// TIA Portal V18 export
FUNCTION "potlife&regenaration" : Void   // FC22, LAD
{ S7_Optimized_Access := 'TRUE' }
VERSION : 0.1
// stored: AutoNumber true, IsIECCheckEnabled false, SetENOAutomatically false, UDAEnableTagReadback false
   VAR_TEMP
      temp2 : Bool;
   END_VAR
   VAR_TEMP   // added for the SCL form of the ladder/FBD networks
      _w1 : Bool;
   END_VAR
BEGIN

REGION Network 1: regeneration selection
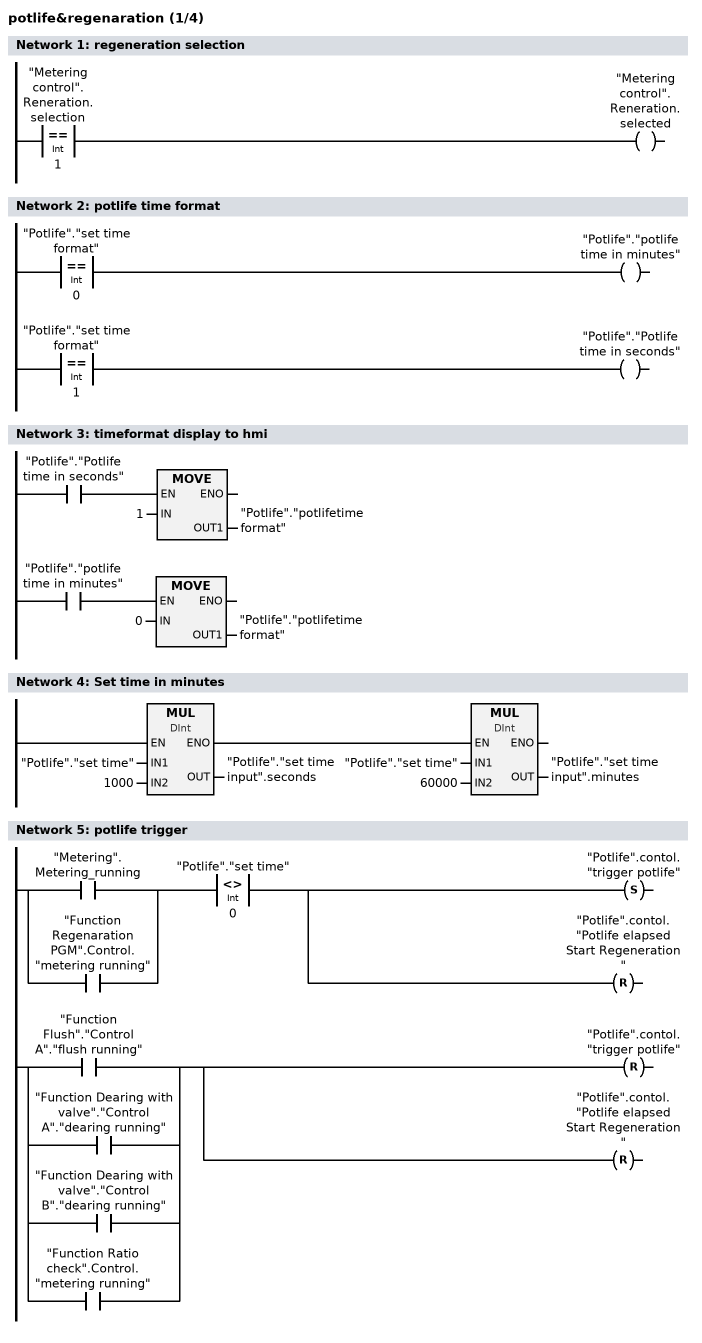
   RUNG wire#powerrail
      { S7_Templates := "SrcType := Int" } EQ_Contact(in1 := "Metering control".Reneration.selection, in2 := 1)
      Coil( "Metering control".Reneration.selected )
   END_RUNG
   // the same network as SCL:
   "Metering control".Reneration.selected := "Metering control".Reneration.selection = 1;
END_REGION

REGION Network 2: potlife time format
   RUNG wire#powerrail
      { S7_Templates := "SrcType := Int" } EQ_Contact(in1 := "Potlife"."set time format", in2 := 0)
      Coil( "Potlife"."potlife time in minutes" )
   END_RUNG
   RUNG wire#powerrail
      { S7_Templates := "SrcType := Int" } EQ_Contact(in1 := "Potlife"."set time format", in2 := 1)
      Coil( "Potlife"."Potlife time in seconds" )
   END_RUNG
   // the same network as SCL:
   "Potlife"."potlife time in minutes" := "Potlife"."set time format" = 0;
   "Potlife"."Potlife time in seconds" := "Potlife"."set time format" = 1;
END_REGION

REGION Network 3: timeformat display to hmi
   RUNG wire#powerrail
      Contact( "Potlife"."Potlife time in seconds" )
      Move(in := 1, out1 => "Potlife"."potlifetime format")
   END_RUNG
   RUNG wire#powerrail
      Contact( "Potlife"."potlife time in minutes" )
      Move(in := 0, out1 => "Potlife"."potlifetime format")
   END_RUNG
   // the same network as SCL:
   IF "Potlife"."Potlife time in seconds" THEN "Potlife"."potlifetime format" := 1; END_IF;
   IF "Potlife"."potlife time in minutes" THEN "Potlife"."potlifetime format" := 0; END_IF;
END_REGION

REGION Network 4: Set time in minutes
   RUNG wire#powerrail
      { S7_Templates := "SrcType := DInt" } Mul(in1 := "Potlife"."set time", in2 := 1000, out => "Potlife"."set time input".seconds)
      { S7_Templates := "SrcType := DInt" } Mul(in1 := "Potlife"."set time", in2 := 60000, out => "Potlife"."set time input".minutes)
   END_RUNG
   // the same network as SCL:
   "Potlife"."set time input".seconds := "Potlife"."set time" * 1000;
   "Potlife"."set time input".minutes := "Potlife"."set time" * 60000;
END_REGION

REGION Network 5: potlife trigger
   RUNG wire#powerrail
      Contact( "Metering".Metering_running )
      wire#w1
      { S7_Templates := "SrcType := Int" } NE_Contact(in1 := "Potlife"."set time", in2 := 0)
      wire#w2
      S_Coil( "Potlife".contol."trigger potlife" )
   END_RUNG
   RUNG wire#powerrail
      Contact( "Function Regenaration PGM".Control."metering running" )
   END_RUNG wire#w1
   RUNG wire#w2
      R_Coil( "Potlife".contol."Potlife elapsed Start Regeneration" )
   END_RUNG
   RUNG wire#powerrail
      Contact( "Function Flush"."Control A"."flush running" )
      wire#w3
      R_Coil( "Potlife".contol."trigger potlife" )
   END_RUNG
   RUNG wire#powerrail
      Contact( "Function Dearing with valve"."Control A"."dearing running" )
   END_RUNG wire#w3
   RUNG wire#powerrail
      Contact( "Function Dearing with valve"."Control B"."dearing running" )
   END_RUNG wire#w3
   RUNG wire#powerrail
      Contact( "Function Ratio check".Control."metering running" )
   END_RUNG wire#w3
   RUNG wire#w3
      R_Coil( "Potlife".contol."Potlife elapsed Start Regeneration" )
   END_RUNG
   // the same network as SCL:
   IF ("Metering".Metering_running OR "Function Regenaration PGM".Control."metering running") AND ("Potlife"."set time" <> 0) THEN
       "Potlife".contol."trigger potlife" := TRUE;
       "Potlife".contol."Potlife elapsed Start Regeneration" := FALSE;
   END_IF;
   IF "Function Flush"."Control A"."flush running" OR "Function Dearing with valve"."Control A"."dearing running" OR "Function Dearing with valve"."Control B"."dearing running" OR "Function Ratio check".Control."metering running" THEN
       "Potlife".contol."trigger potlife" := FALSE;
       "Potlife".contol."Potlife elapsed Start Regeneration" := FALSE;
   END_IF;
END_REGION

REGION Network 6
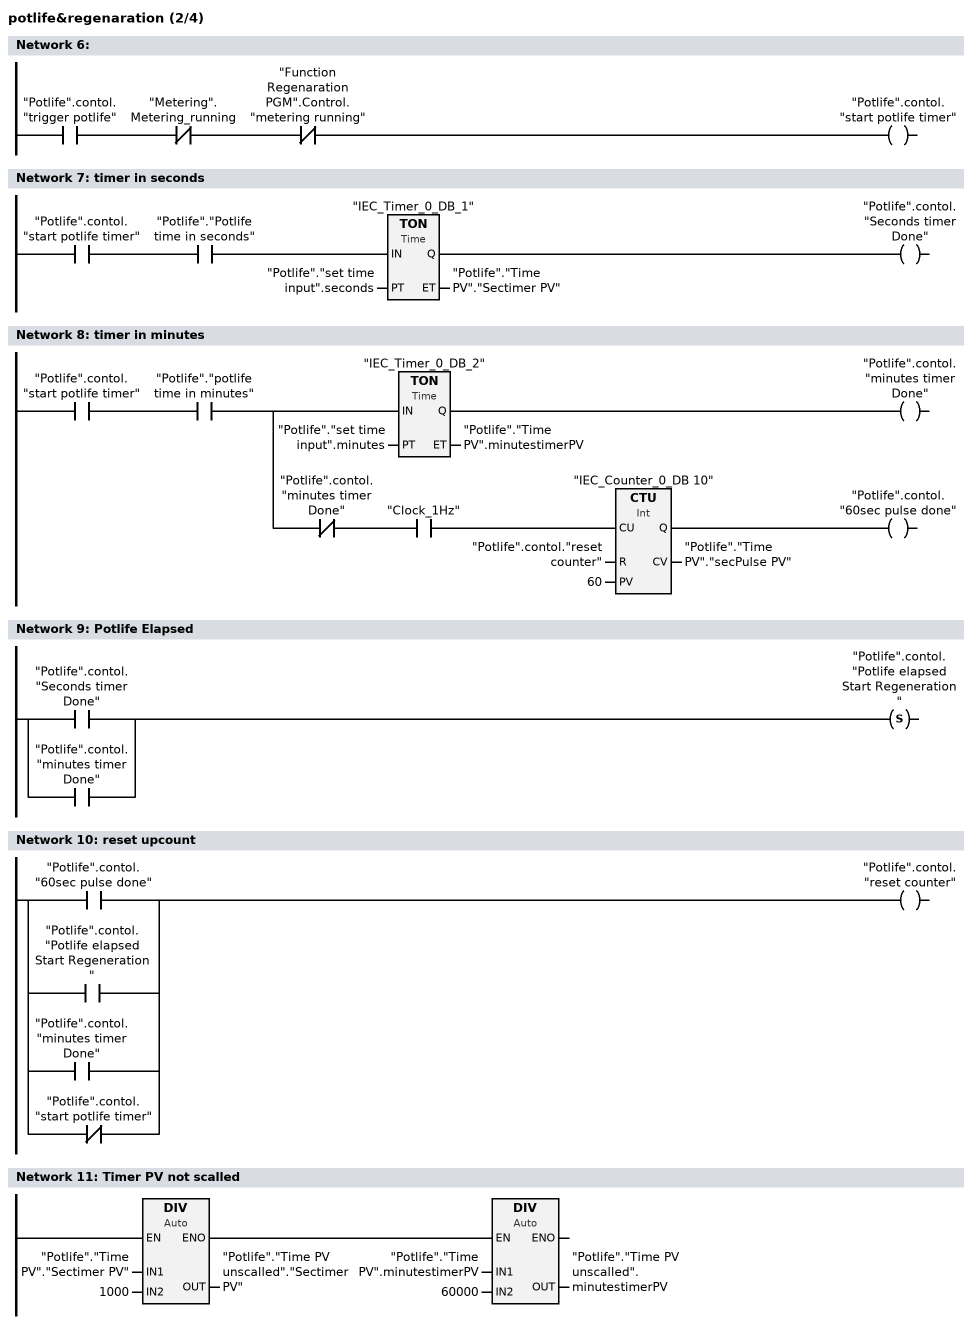
   RUNG wire#powerrail
      Contact( "Potlife".contol."trigger potlife" )
      I_Contact( "Metering".Metering_running )
      I_Contact( "Function Regenaration PGM".Control."metering running" )
      Coil( "Potlife".contol."start potlife timer" )
   END_RUNG
   // the same network as SCL:
   "Potlife".contol."start potlife timer" := "Potlife".contol."trigger potlife" AND NOT "Metering".Metering_running AND NOT "Function Regenaration PGM".Control."metering running";
END_REGION

REGION Network 7: timer in seconds
   RUNG wire#powerrail
      Contact( "Potlife".contol."start potlife timer" )
      Contact( "Potlife"."Potlife time in seconds" )
      { S7_Templates := "time_type := Time" } "IEC_Timer_0_DB_1".TON(pt := "Potlife"."set time input".seconds, et => "Potlife"."Time PV"."Sectimer PV")
      Coil( "Potlife".contol."Seconds timer Done" )
   END_RUNG
   // the same network as SCL:
   "IEC_Timer_0_DB_1".TON(IN := "Potlife".contol."start potlife timer" AND "Potlife"."Potlife time in seconds",
                          PT := "Potlife"."set time input".seconds,
                          ET => "Potlife"."Time PV"."Sectimer PV");
   "Potlife".contol."Seconds timer Done" := "IEC_Timer_0_DB_1".Q;
END_REGION

REGION Network 8: timer in minutes
   RUNG wire#powerrail
      Contact( "Potlife".contol."start potlife timer" )
      Contact( "Potlife"."potlife time in minutes" )
      wire#w1
      { S7_Templates := "time_type := Time" } "IEC_Timer_0_DB_2".TON(pt := "Potlife"."set time input".minutes, et => "Potlife"."Time PV".minutestimerPV)
      Coil( "Potlife".contol."minutes timer Done" )
   END_RUNG
   RUNG wire#w1
      I_Contact( "Potlife".contol."minutes timer Done" )
      Contact( "Clock_1Hz" )
      { S7_Templates := "value_type := Int" } "IEC_Counter_0_DB 10".CTU(r := "Potlife".contol."reset counter", pv := 60, cv => "Potlife"."Time PV"."secPulse PV")
      Coil( "Potlife".contol."60sec pulse done" )
   END_RUNG
   // the same network as SCL:
   #_w1 := "Potlife".contol."start potlife timer" AND "Potlife"."potlife time in minutes";
   "IEC_Timer_0_DB_2".TON(IN := #_w1,
                          PT := "Potlife"."set time input".minutes,
                          ET => "Potlife"."Time PV".minutestimerPV);
   "Potlife".contol."minutes timer Done" := "IEC_Timer_0_DB_2".Q;
   "IEC_Counter_0_DB 10".CTU(CU := #_w1 AND NOT "Potlife".contol."minutes timer Done" AND "Clock_1Hz",
                           R := "Potlife".contol."reset counter",
                           PV := 60,
                           CV => "Potlife"."Time PV"."secPulse PV");
   "Potlife".contol."60sec pulse done" := "IEC_Counter_0_DB 10".Q;
END_REGION

REGION Network 9: Potlife Elapsed
   RUNG wire#powerrail
      Contact( "Potlife".contol."Seconds timer Done" )
      wire#w1
      S_Coil( "Potlife".contol."Potlife elapsed Start Regeneration" )
   END_RUNG
   RUNG wire#powerrail
      Contact( "Potlife".contol."minutes timer Done" )
   END_RUNG wire#w1
   // the same network as SCL:
   IF "Potlife".contol."Seconds timer Done" OR "Potlife".contol."minutes timer Done" THEN
       "Potlife".contol."Potlife elapsed Start Regeneration" := TRUE;
   END_IF;
END_REGION

REGION Network 10: reset upcount
   RUNG wire#powerrail
      Contact( "Potlife".contol."60sec pulse done" )
      wire#w1
      Coil( "Potlife".contol."reset counter" )
   END_RUNG
   RUNG wire#powerrail
      Contact( "Potlife".contol."Potlife elapsed Start Regeneration" )
   END_RUNG wire#w1
   RUNG wire#powerrail
      Contact( "Potlife".contol."minutes timer Done" )
   END_RUNG wire#w1
   RUNG wire#powerrail
      I_Contact( "Potlife".contol."start potlife timer" )
   END_RUNG wire#w1
   // the same network as SCL:
   "Potlife".contol."reset counter" := "Potlife".contol."60sec pulse done" OR "Potlife".contol."Potlife elapsed Start Regeneration" OR "Potlife".contol."minutes timer Done" OR NOT "Potlife".contol."start potlife timer";
END_REGION

REGION Network 11: Timer PV not scalled
   RUNG wire#powerrail
      Div(in1 := "Potlife"."Time PV"."Sectimer PV", in2 := 1000, out => "Potlife"."Time PV unscalled"."Sectimer PV")
      Div(in1 := "Potlife"."Time PV".minutestimerPV, in2 := 60000, out => "Potlife"."Time PV unscalled".minutestimerPV)
   END_RUNG
   // the same network as SCL:
   "Potlife"."Time PV unscalled"."Sectimer PV" := "Potlife"."Time PV"."Sectimer PV" / 1000;
   "Potlife"."Time PV unscalled".minutestimerPV := "Potlife"."Time PV".minutestimerPV / 60000;
END_REGION

REGION Network 12: run time down count
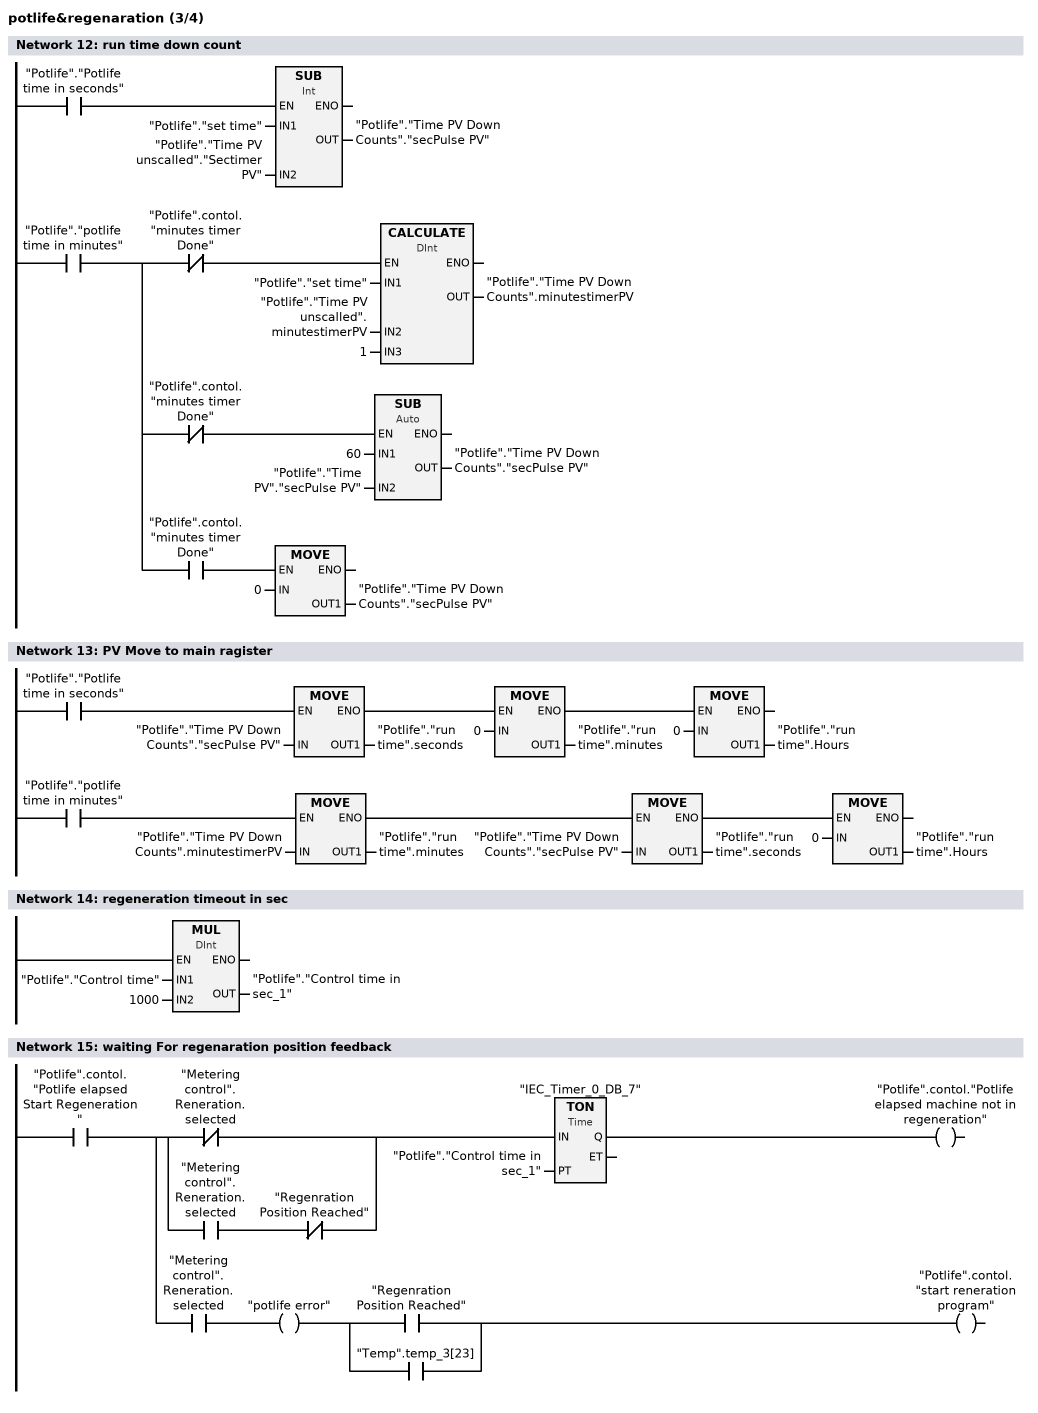
   RUNG wire#powerrail
      Contact( "Potlife"."Potlife time in seconds" )
      { S7_Templates := "SrcType := Int" } Sub(in1 := "Potlife"."set time", in2 := "Potlife"."Time PV unscalled"."Sectimer PV", out => "Potlife"."Time PV Down Counts"."secPulse PV")
   END_RUNG
   RUNG wire#powerrail
      Contact( "Potlife"."potlife time in minutes" )
      wire#w1
      I_Contact( "Potlife".contol."minutes timer Done" )
      { S7_Templates := "SrcType := DInt"; S7_Expression := "IN1-IN2-IN3" } Calculate(in1 := "Potlife"."set time", in2 := "Potlife"."Time PV unscalled".minutestimerPV, in3 := 1, out => "Potlife"."Time PV Down Counts".minutestimerPV)
   END_RUNG
   RUNG wire#w1
      I_Contact( "Potlife".contol."minutes timer Done" )
      Sub(in1 := 60, in2 := "Potlife"."Time PV"."secPulse PV", out => "Potlife"."Time PV Down Counts"."secPulse PV")
   END_RUNG
   RUNG wire#w1
      Contact( "Potlife".contol."minutes timer Done" )
      Move(in := 0, out1 => "Potlife"."Time PV Down Counts"."secPulse PV")
   END_RUNG
   // the same network as SCL:
   IF "Potlife"."Potlife time in seconds" THEN
       "Potlife"."Time PV Down Counts"."secPulse PV" := "Potlife"."set time" - "Potlife"."Time PV unscalled"."Sectimer PV";
   END_IF;
   IF "Potlife"."potlife time in minutes" AND NOT "Potlife".contol."minutes timer Done" THEN
       "Potlife"."Time PV Down Counts".minutestimerPV := "Potlife"."set time"-"Potlife"."Time PV unscalled".minutestimerPV-1;
       "Potlife"."Time PV Down Counts"."secPulse PV" := 60 - "Potlife"."Time PV"."secPulse PV";
   END_IF;
   IF "Potlife"."potlife time in minutes" AND "Potlife".contol."minutes timer Done" THEN
       "Potlife"."Time PV Down Counts"."secPulse PV" := 0;
   END_IF;
END_REGION

REGION Network 13: PV Move to main ragister
   RUNG wire#powerrail
      Contact( "Potlife"."Potlife time in seconds" )
      Move(in := "Potlife"."Time PV Down Counts"."secPulse PV", out1 => "Potlife"."run time".seconds)
      Move(in := 0, out1 => "Potlife"."run time".minutes)
      Move(in := 0, out1 => "Potlife"."run time".Hours)
   END_RUNG
   RUNG wire#powerrail
      Contact( "Potlife"."potlife time in minutes" )
      Move(in := "Potlife"."Time PV Down Counts".minutestimerPV, out1 => "Potlife"."run time".minutes)
      Move(in := "Potlife"."Time PV Down Counts"."secPulse PV", out1 => "Potlife"."run time".seconds)
      Move(in := 0, out1 => "Potlife"."run time".Hours)
   END_RUNG
   // the same network as SCL:
   IF "Potlife"."Potlife time in seconds" THEN
       "Potlife"."run time".seconds := "Potlife"."Time PV Down Counts"."secPulse PV";
       "Potlife"."run time".minutes := 0;
       "Potlife"."run time".Hours := 0;
   END_IF;
   IF "Potlife"."potlife time in minutes" THEN
       "Potlife"."run time".minutes := "Potlife"."Time PV Down Counts".minutestimerPV;
       "Potlife"."run time".seconds := "Potlife"."Time PV Down Counts"."secPulse PV";
       "Potlife"."run time".Hours := 0;
   END_IF;
END_REGION

REGION Network 14: regeneration timeout in sec
   RUNG wire#powerrail
      { S7_Templates := "SrcType := DInt" } Mul(in1 := "Potlife"."Control time", in2 := 1000, out => "Potlife"."Control time in sec_1")
   END_RUNG
   // the same network as SCL:
   "Potlife"."Control time in sec_1" := "Potlife"."Control time" * 1000;
END_REGION

REGION Network 15: waiting For regenaration position feedback
   RUNG wire#powerrail
      Contact( "Potlife".contol."Potlife elapsed Start Regeneration" )
      wire#w1
      I_Contact( "Metering control".Reneration.selected )
      wire#w2
      { S7_Templates := "time_type := Time" } "IEC_Timer_0_DB_7".TON(pt := "Potlife"."Control time in sec_1", et =>)
      Coil( "Potlife".contol."Potlife elapsed machine not in regeneration" )
   END_RUNG
   RUNG wire#w1
      Contact( "Metering control".Reneration.selected )
      I_Contact( "Regenration Position Reached" )
   END_RUNG wire#w2
   RUNG wire#w1
      Contact( "Metering control".Reneration.selected )
      Coil( "potlife error" )
      wire#w3
      Contact( "Regenration Position Reached" )
      wire#w4
      Coil( "Potlife".contol."start reneration program" )
   END_RUNG
   RUNG wire#w3
      Contact( "Temp".temp_3[23] )
   END_RUNG wire#w4
   // the same network as SCL:
   "IEC_Timer_0_DB_7".TON(IN := "Potlife".contol."Potlife elapsed Start Regeneration" AND (NOT "Metering control".Reneration.selected OR ("Metering control".Reneration.selected AND NOT "Regenration Position Reached")),
                          PT := "Potlife"."Control time in sec_1");
   "Potlife".contol."Potlife elapsed machine not in regeneration" := "IEC_Timer_0_DB_7".Q;
   "potlife error" := "Potlife".contol."Potlife elapsed Start Regeneration" AND "Metering control".Reneration.selected;
   "Potlife".contol."start reneration program" := "potlife error" AND ("Regenration Position Reached" OR "Temp".temp_3[23]);
END_REGION

REGION Network 16: Selecting regeneration program
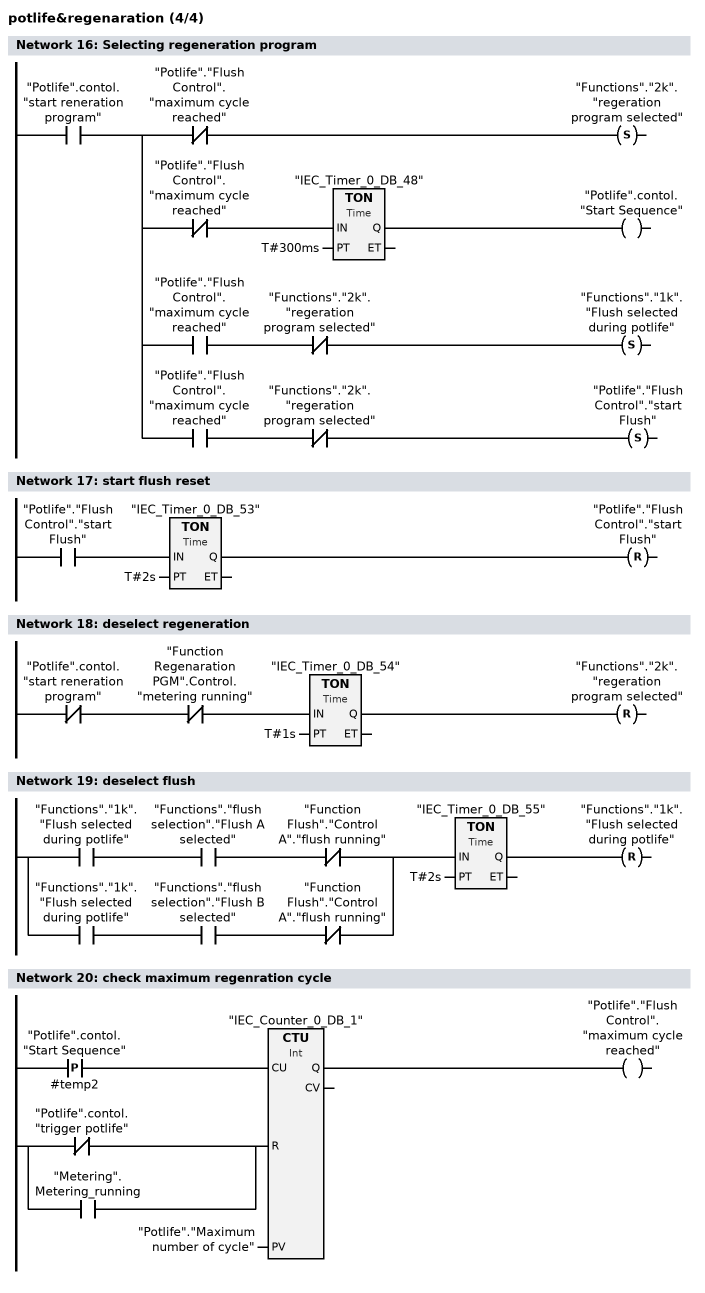
   RUNG wire#powerrail
      Contact( "Potlife".contol."start reneration program" )
      wire#w1
      I_Contact( "Potlife"."Flush Control"."maximum cycle reached" )
      S_Coil( "Functions"."2k"."regeration program selected" )
   END_RUNG
   RUNG wire#w1
      I_Contact( "Potlife"."Flush Control"."maximum cycle reached" )
      { S7_Templates := "time_type := Time" } "IEC_Timer_0_DB_48".TON(pt := T#300ms, et =>)
      Coil( "Potlife".contol."Start Sequence" )
   END_RUNG
   RUNG wire#w1
      Contact( "Potlife"."Flush Control"."maximum cycle reached" )
      I_Contact( "Functions"."2k"."regeration program selected" )
      S_Coil( "Functions"."1k"."Flush selected during potlife" )
   END_RUNG
   RUNG wire#w1
      Contact( "Potlife"."Flush Control"."maximum cycle reached" )
      I_Contact( "Functions"."2k"."regeration program selected" )
      S_Coil( "Potlife"."Flush Control"."start Flush" )
   END_RUNG
   // the same network as SCL:
   IF "Potlife".contol."start reneration program" AND NOT "Potlife"."Flush Control"."maximum cycle reached" THEN
       "Functions"."2k"."regeration program selected" := TRUE;
   END_IF;
   "IEC_Timer_0_DB_48".TON(IN := "Potlife".contol."start reneration program" AND NOT "Potlife"."Flush Control"."maximum cycle reached",
                           PT := T#300ms);
   "Potlife".contol."Start Sequence" := "IEC_Timer_0_DB_48".Q;
   IF "Potlife".contol."start reneration program" AND "Potlife"."Flush Control"."maximum cycle reached" AND NOT "Functions"."2k"."regeration program selected" THEN
       "Functions"."1k"."Flush selected during potlife" := TRUE;
       "Potlife"."Flush Control"."start Flush" := TRUE;
   END_IF;
END_REGION

REGION Network 17: start flush reset
   RUNG wire#powerrail
      Contact( "Potlife"."Flush Control"."start Flush" )
      { S7_Templates := "time_type := Time" } "IEC_Timer_0_DB_53".TON(pt := T#2s, et =>)
      R_Coil( "Potlife"."Flush Control"."start Flush" )
   END_RUNG
   // the same network as SCL:
   "IEC_Timer_0_DB_53".TON(IN := "Potlife"."Flush Control"."start Flush", PT := T#2s);
   IF "IEC_Timer_0_DB_53".Q THEN "Potlife"."Flush Control"."start Flush" := FALSE; END_IF;
END_REGION

REGION Network 18: deselect regeneration
   RUNG wire#powerrail
      I_Contact( "Potlife".contol."start reneration program" )
      I_Contact( "Function Regenaration PGM".Control."metering running" )
      { S7_Templates := "time_type := Time" } "IEC_Timer_0_DB_54".TON(pt := T#1s, et =>)
      R_Coil( "Functions"."2k"."regeration program selected" )
   END_RUNG
   // the same network as SCL:
   "IEC_Timer_0_DB_54".TON(IN := NOT "Potlife".contol."start reneration program" AND NOT "Function Regenaration PGM".Control."metering running",
                           PT := T#1s);
   IF "IEC_Timer_0_DB_54".Q THEN "Functions"."2k"."regeration program selected" := FALSE; END_IF;
END_REGION

REGION Network 19: deselect flush
   RUNG wire#powerrail
      Contact( "Functions"."1k"."Flush selected during potlife" )
      Contact( "Functions"."flush selection"."Flush A selected" )
      I_Contact( "Function Flush"."Control A"."flush running" )
      wire#w1
      { S7_Templates := "time_type := Time" } "IEC_Timer_0_DB_55".TON(pt := T#2s, et =>)
      R_Coil( "Functions"."1k"."Flush selected during potlife" )
   END_RUNG
   RUNG wire#powerrail
      Contact( "Functions"."1k"."Flush selected during potlife" )
      Contact( "Functions"."flush selection"."Flush B selected" )
      I_Contact( "Function Flush"."Control A"."flush running" )
   END_RUNG wire#w1
   // the same network as SCL:
   "IEC_Timer_0_DB_55".TON(IN := ("Functions"."1k"."Flush selected during potlife" AND "Functions"."flush selection"."Flush A selected" AND NOT "Function Flush"."Control A"."flush running") OR ("Functions"."1k"."Flush selected during potlife" AND "Functions"."flush selection"."Flush B selected" AND NOT "Function Flush"."Control A"."flush running"),
                           PT := T#2s);
   IF "IEC_Timer_0_DB_55".Q THEN "Functions"."1k"."Flush selected during potlife" := FALSE; END_IF;
END_REGION

REGION Network 20: check maximum regenration cycle
   RUNG wire#powerrail
      P_Contact(operand := "Potlife".contol."Start Sequence", bit := #temp2)
      { S7_Templates := "value_type := Int" } "IEC_Counter_0_DB_1".CTU(r := wire#w1, pv := "Potlife"."Maximum number of cycle", cv =>)
      Coil( "Potlife"."Flush Control"."maximum cycle reached" )
   END_RUNG
   RUNG wire#powerrail
      I_Contact( "Potlife".contol."trigger potlife" )
   END_RUNG wire#w1
   RUNG wire#powerrail
      Contact( "Metering".Metering_running )
   END_RUNG wire#w1
   // the same network as SCL:
   #_w1 := "Potlife".contol."Start Sequence" AND NOT #temp2;   // rising edge of "Potlife".contol."Start Sequence"
   #temp2 := "Potlife".contol."Start Sequence";
   "IEC_Counter_0_DB_1".CTU(CU := #_w1,
                           R := NOT "Potlife".contol."trigger potlife" OR "Metering".Metering_running,
                           PV := "Potlife"."Maximum number of cycle");
   "Potlife"."Flush Control"."maximum cycle reached" := "IEC_Counter_0_DB_1".Q;
END_REGION
END_FUNCTION
